% RSLogix 500 project PLC Automated Sensor Calibration.RSS, saved by version 8.30.00.16 %
PROJECT "UNTITLED"    % processor: Bul.1763 MicroLogix 1100 Series B %

PROGRAM FILES
  LAD 2 "MAIN"  3 rungs
  LAD 3 "IO"  3 rungs
  LAD 4 "CONTROLS"  8 rungs

DATA FILES
  O0 OUTPUT  4 elements
  I1 INPUT  6 elements
  S2 STATUS  66 elements
  B3 BINARY  1 elements
  T4 TIMER  4 elements
  C5 COUNTER  1 elements
  R6 CONTROL  1 elements
  N7 INTEGER  11 elements
  F8 FLOAT  2 elements

LADDER 2 "MAIN"
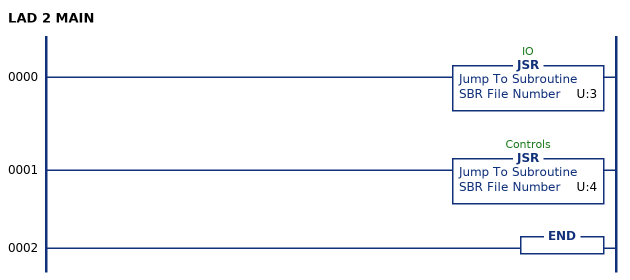
% Rung: 0 %
SOR JSR U:3 EOR
%   U:3  "IO" %
% Rung: 1 %
SOR JSR U:4 EOR
%   U:4  "Controls" %
% Rung: 2 %
SOR END EOR

LADDER 3 "IO"
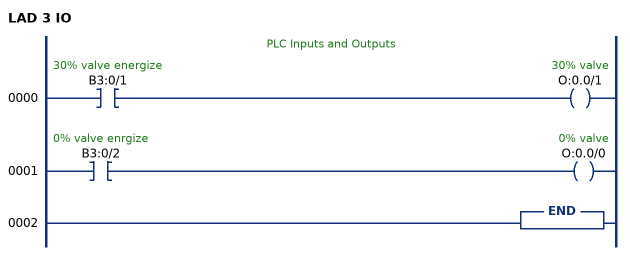
% Rung: 0 %
% PLC Inputs and Outputs %
SOR XIC B3:0/1 OTE O:0.0/1 EOR
%   B3:0/1  "30% valve energize" %
%   O:0.0/1  "30% valve" %
% Rung: 1 %
SOR XIC B3:0/2 OTE O:0.0/0 EOR
%   B3:0/2  "0% valve enrgize" %
%   O:0.0/0  "0% valve" %
% Rung: 2 %
SOR END EOR

LADDER 4 "CONTROLS"
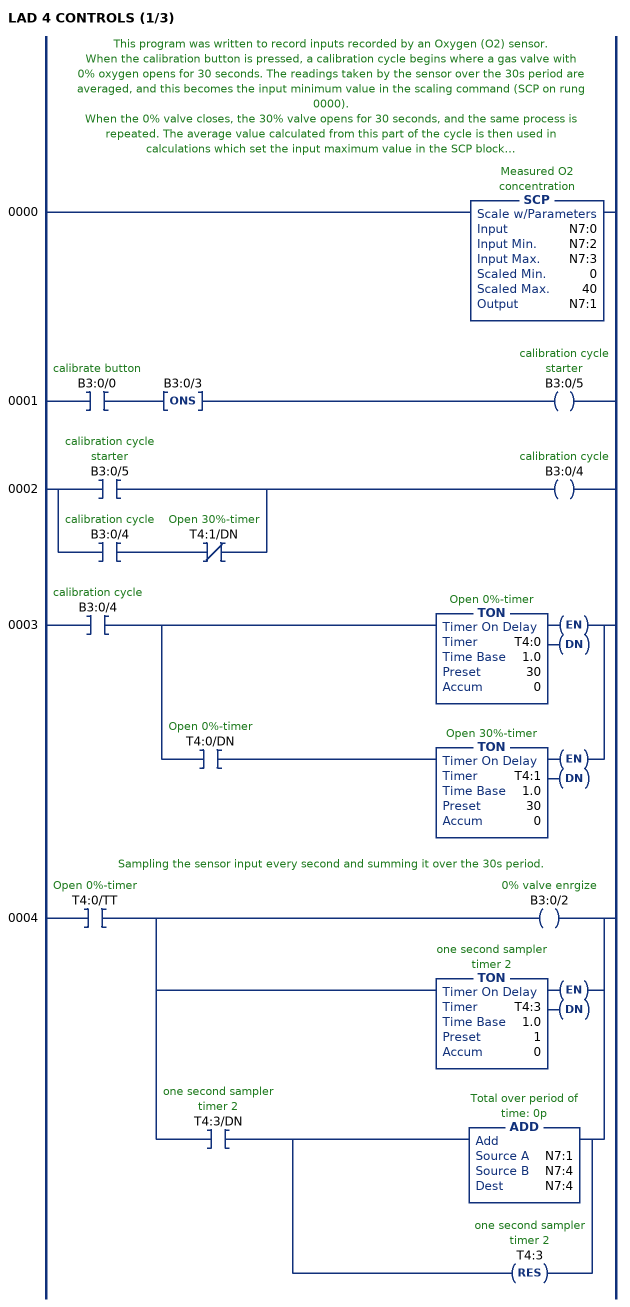
% Rung: 0 %
% This program was written to record inputs recorded by an Oxygen (O2) sensor.
% When the calibration button is pressed, a calibration cycle begins where a gas valve with 0% oxygen opens for 30 seconds. The readings taken by the sensor over the 30s period are averaged, and this becomes the input minimum value in the scaling command (SCP on rung 0000).
% When the 0% valve closes, the 30% valve opens for 30 seconds, and the same process is repeated. The average value calculated from this part of the cycle is then used in calculations which set the input maximum value in the SCP block.
% When the 30% valve is closed, the calibration cycle ends. %
SOR SCP N7:0 N7:2 N7:3 0 40 N7:1 EOR
%   N7:0  "O2 sensor signal input" %
%   N7:2  "Input Min" %
%   N7:3  "Input Max" %
%   N7:1  "Measured O2 concentration" %
% Rung: 1 %
SOR XIC B3:0/0 ONS B3:0/3 OTE B3:0/5 EOR
%   B3:0/0  "calibrate button" %
%   B3:0/5  "calibration cycle starter" %
% Rung: 2 %
SOR BST XIC B3:0/5 NXB XIC B3:0/4 XIO T4:1/DN BND OTE B3:0/4 EOR
%   B3:0/5  "calibration cycle starter" %
%   B3:0/4  "calibration cycle" %
%   T4:1  "Open 30%-timer" %
% Rung: 3 %
SOR XIC B3:0/4 BST TON T4:0 1.0 30 0 NXB XIC T4:0/DN TON T4:1 1.0 30 0 BND EOR
%   B3:0/4  "calibration cycle" %
%   T4:0  "Open 0%-timer" %
%   T4:1  "Open 30%-timer" %
% Rung: 4 %
% Sampling the sensor input every second and summing it over the 30s period. %
SOR XIC T4:0/TT BST OTE B3:0/2 NXB TON T4:3 1.0 1 0 NXB XIC T4:3/DN BST ADD N7:1 N7:4 N7:4 NXB RES T4:3 BND BND EOR
%   T4:0  "Open 0%-timer" %
%   B3:0/2  "0% valve enrgize" %
%   T4:3  "one second sampler timer 2" %
%   N7:1  "Measured O2 concentration" %
%   N7:4  "Total over period of time: 0p" %

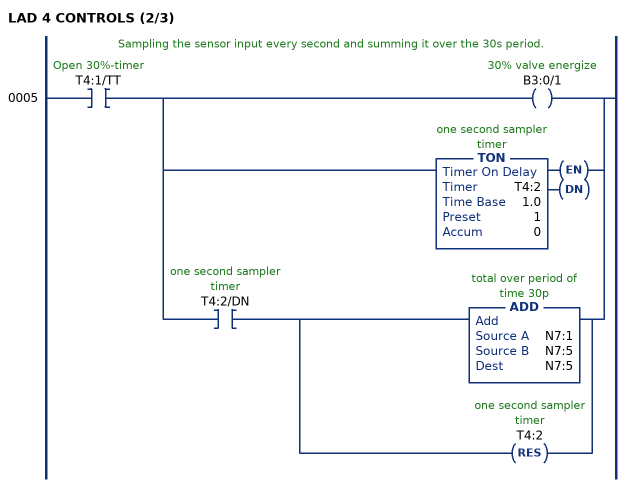
% Rung: 5 %
% Sampling the sensor input every second and summing it over the 30s period. %
SOR XIC T4:1/TT BST OTE B3:0/1 NXB TON T4:2 1.0 1 0 NXB XIC T4:2/DN BST ADD N7:1 N7:5 N7:5 NXB RES T4:2 BND BND EOR
%   T4:1  "Open 30%-timer" %
%   B3:0/1  "30% valve energize" %
%   T4:2  "one second sampler timer" %
%   N7:1  "Measured O2 concentration" %
%   N7:5  "total over period of time 30p" %

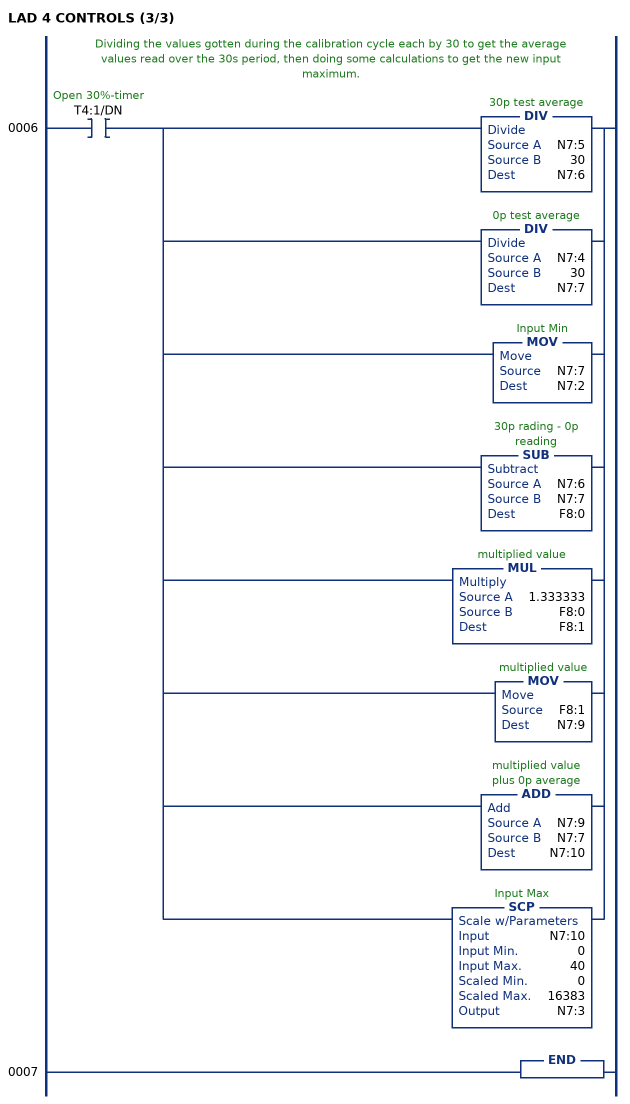
% Rung: 6 %
% Dividing the values gotten during the calibration cycle each by 30 to get the average values read over the 30s period, then doing some calculations to get the new input maximum. %
SOR XIC T4:1/DN BST DIV N7:5 30 N7:6 NXB DIV N7:4 30 N7:7 NXB MOV N7:7 N7:2 NXB SUB N7:6 N7:7 F8:0 NXB MUL 1.333333 F8:0 F8:1 NXB MOV F8:1 N7:9 NXB ADD N7:9 N7:7 N7:10 NXB SCP N7:10 0 40 0 16383 N7:3 BND EOR
%   T4:1  "Open 30%-timer" %
%   N7:5  "total over period of time 30p" %
%   N7:6  "30p test average" %
%   N7:4  "Total over period of time: 0p" %
%   N7:7  "0p test average" %
%   N7:2  "Input Min" %
%   F8:0  "30p rading - 0p reading" %
%   F8:1  "multiplied value" %
%   N7:9  "multiplied value" %
%   N7:10  "multiplied value plus 0p average" %
%   N7:3  "Input Max" %
% Rung: 7 %
SOR END EOR

OTHER DOCUMENTED ADDRESSES
  B3  

DATA TABLE (non-zero values as saved)
DATA B3
% B3:0 % 0X0049
DATA T4
% .PRE .ACC %
% T4:0 % 30 0
% T4:1 % 30 0
% T4:2 % 1 0
% T4:3 % 1 0
DATA N7
% N7:0 % 14633 30 0 19250 0 1044 35 0 0 47
% N7:10 % 47
DATA F8
% F8:0 % 35 46.66666
